# B&R Automation Studio project OPSULab3
Automation Studio 4.5.2.102

## Configuration Config1

### Task classes (Cpu.sw)
```
Cyclic#1:
  ncsdcctrl <- ncsdcctrl.prg
Cyclic#4:
  Program <- Program.prg
NcDataObjects: acp10etxen <- acp10etxen.dob, gAxis01a <- gAxis01obj.gAxis01a.dob, gAxis01i <- gAxis01obj.gAxis01i.dob
VcDataObjects: Visu <- Visu.dob
Libraries: Acp10man, Acp10par, NcGlobal, Acp10sdc, AsBrStr, Acp10_MC, brsystem, sys_lib, runtime, Library
```

### IoMap.iom - 4PP065_0571_P74/IoMap.iom
```iecst
VAR_CONFIG
	Cyclic#1.gAxis01_DrvIf.iLifeCnt AT %IB."8I64xxxxxxx.00x-1".SDC_LifeCnt;
	Cyclic#1.gAxis01_DrvIf.iDrvOK AT %IX."8I64xxxxxxx.00x-1".ETAD_Input_Bool_02;
	Cyclic#1.gAxis01_DrvIf.oSetTime AT %QW."8I64xxxxxxx.00x-1".SDC_SetTime;
	Cyclic#1.::speed AT %QW."8I64xxxxxxx.00x-1".LFRD_Output;
	Cyclic#1.gAxis01_DiDoIf.iLifeCntDriveReady AT %IB."8I64xxxxxxx.00x-1".SDC_LifeCnt;
	Cyclic#1.gAxis01_DiDoIf.iLifeCntDriveEnable AT %IB."8I64xxxxxxx.00x-1".SDC_LifeCnt;
	Cyclic#1.gAxis01_DiDoIf.oDriveEnable AT %QX."8I64xxxxxxx.00x-1".CMDD_Output_Bool_00;
	Cyclic#1.gAxis01_ModuleOk AT %QX."8I64xxxxxxx.00x-1".CMDD_Output_Bool_01;
	Cyclic#1.gAxis01_ModuleOk AT %QX."8I64xxxxxxx.00x-1".CMDD_Output_Bool_02;
	Cyclic#1.gAxis01_ModuleOk AT %IX."8I64xxxxxxx.00x-1".ModuleOk;
	Cyclic#1.gAxis01_DiDoIf.oDriveEnable AT %QX."8I64xxxxxxx.00x-1".CMDD_Output_Bool_03;
	Cyclic#1.gAxis01_DiDoIf.iDriveReady AT %IX."8I64xxxxxxx.00x-1".ETAD_Input_Bool_02;
	::EVIRD.STATE AT %IW."8I64xxxxxxx.00x-1".ETAD_Input;
	::EVIRD.CMD AT %QW."8I64xxxxxxx.00x-1".CMDD_Output;
END_VAR
```

## Logical view

Binary libraries used (declarations not repeated): Library

### Global.var - Global variables
```iecst
VAR
	gAxis01 : ACP10AXIS_typ;
	gAxis01_HW : SdcHwCfg_typ := (0);
	gAxis01_DrvIf : SdcDrvIf16_typ := (0);
	gAxis01_DiDoIf : SdcDiDoIf_typ := (0);
	gAxis01_ModuleOk : BOOL := 0;
	speed : INT := 500;
	EVIRD : DRIVE;
	OnButton : BOOL;
END_VAR
```

### Package Logical/Libraries - Global libraries

- Visualisation Logical/Visu (not shown)

Listed in the project but not available here: Logical/Global.typ, Logical/acp10etxen, Logical/ncsdcctrl, Logical/gAxis01obj, Logical/Program
